// TwinCAT 3 PLC project EDA
// ProgramVersion: 3.1.4024.0
// libraries:
//   Tc2_Standard, * (Beckhoff Automation GmbH)
//   Tc2_System, * (Beckhoff Automation GmbH)
//   Tc3_Module, * (Beckhoff Automation GmbH)
// project tree:
//   GVLs/ GVL.TcGVL
//   / PlcTask.TcTTO
//   POUs/ MAIN.TcPOU
// real-time tasks:
//   TASK PlcTask: cycle T#10ms, priority 20, ADS port 350
// I/O:
//   DEVICE Device 1 (EtherCAT), AmsNetId 5.119.159.52.2.1
//     Term 1 (EK1200) [EK1200-5000 EtherCAT Power supply (2A E-Bus)]
//       Term 2 (EL3443) [EL3443 3Ch. Power Measuring]
//       Term 3 (EL9011) [EL9011 End Terminal]
// variable links:
//   EDA/EDA Instance <-> Device 1 (EtherCAT)/Term 1 (EK1200)/Term 2 (EL3443)
//     PlcTask Inputs/GVL.EL3443.MDP5001_341_Input/MDP5001_341_L1_Basic_Current <-> L1 Basic/Current
//     PlcTask Inputs/GVL.EL3443.MDP5001_341_Input/MDP5001_341_L1_Basic_Voltage <-> L1 Basic/Voltage
//     PlcTask Inputs/GVL.EL3443.MDP5001_341_Input/MDP5001_341_L1_Power_Active_Power <-> L1 Power/Active Power
//     PlcTask Inputs/GVL.EL3443.MDP5001_341_Input/MDP5001_341_L1_Power_Apparent_Power <-> L1 Power/Apparent Power
//     PlcTask Inputs/GVL.EL3443.MDP5001_341_Input/MDP5001_341_L1_Power_Power_Factor <-> L1 Power/Power Factor
//     PlcTask Inputs/GVL.EL3443.MDP5001_341_Input/MDP5001_341_L1_Power_Reactive_Power <-> L1 Power/Reactive Power
//     PlcTask Inputs/GVL.EL3443.MDP5001_341_Input/MDP5001_341_L1_Status_Current_Guard_Error <-> L1 Status/Current Guard Error
//     PlcTask Inputs/GVL.EL3443.MDP5001_341_Input/MDP5001_341_L1_Status_Current_Guard_Warning <-> L1 Status/Current Guard Warning
//     PlcTask Inputs/GVL.EL3443.MDP5001_341_Input/MDP5001_341_L1_Status_Inaccurate_Current <-> L1 Status/Inaccurate Current
//     PlcTask Inputs/GVL.EL3443.MDP5001_341_Input/MDP5001_341_L1_Status_Inaccurate_Voltage <-> L1 Status/Inaccurate Voltage
//     PlcTask Inputs/GVL.EL3443.MDP5001_341_Input/MDP5001_341_L1_Status_Overcurrent <-> L1 Status/Overcurrent
//     PlcTask Inputs/GVL.EL3443.MDP5001_341_Input/MDP5001_341_L1_Status_Overvoltage <-> L1 Status/Overvoltage
//     PlcTask Inputs/GVL.EL3443.MDP5001_341_Input/MDP5001_341_L1_Status_TxPDO_Toggle <-> L1 Status/TxPDO Toggle
//     PlcTask Inputs/GVL.EL3443.MDP5001_341_Input/MDP5001_341_L1_Status_Voltage_Guard_Error <-> L1 Status/Voltage Guard Error
//     PlcTask Inputs/GVL.EL3443.MDP5001_341_Input/MDP5001_341_L1_Status_Voltage_Guard_Warning <-> L1 Status/Voltage Guard Warning
//     PlcTask Inputs/GVL.EL3443.MDP5001_341_Input/MDP5001_341_L1_Status_Voltage_Sign_Bit <-> L1 Status/Voltage Sign Bit
//     PlcTask Inputs/GVL.EL3443.MDP5001_341_Input/MDP5001_341_L1_Timing_Voltage_Last_Zero_Crossing <-> L1 Timing/Voltage Last Zero Crossing
//     PlcTask Inputs/GVL.EL3443.MDP5001_341_Input/MDP5001_341_Total_Basic_Calculated_Neutral_Line_Current <-> Total Basic/Calculated Neutral Line Current
//     PlcTask Inputs/GVL.EL3443.MDP5001_341_Input/MDP5001_341_Total_Basic_Frequency <-> Total Basic/Frequency
//     PlcTask Inputs/GVL.EL3443.MDP5001_341_Input/MDP5001_341_Total_Basic_Power_Factor <-> Total Basic/Power Factor
//     PlcTask Inputs/GVL.EL3443.MDP5001_341_Input/MDP5001_341_Total_Status_Active_Power_Guard_Error <-> Total Status/Active Power Guard Error
//     PlcTask Inputs/GVL.EL3443.MDP5001_341_Input/MDP5001_341_Total_Status_Active_Power_Guard_Warning <-> Total Status/Active Power Guard Warning
//     PlcTask Inputs/GVL.EL3443.MDP5001_341_Input/MDP5001_341_Total_Status_Apparent_Power_Guard_Error <-> Total Status/Apparent Power Guard Error
//     PlcTask Inputs/GVL.EL3443.MDP5001_341_Input/MDP5001_341_Total_Status_Apparent_Power_Guard_Warning <-> Total Status/Apparent Power Guard Warning
//     PlcTask Inputs/GVL.EL3443.MDP5001_341_Input/MDP5001_341_Total_Status_Frequency_Guard_Error <-> Total Status/Frequency Guard Error
//     PlcTask Inputs/GVL.EL3443.MDP5001_341_Input/MDP5001_341_Total_Status_Frequency_Guard_Warning <-> Total Status/Frequency Guard Warning
//     PlcTask Inputs/GVL.EL3443.MDP5001_341_Input/MDP5001_341_Total_Status_Grid_Direction <-> Total Status/Grid Direction
//     PlcTask Inputs/GVL.EL3443.MDP5001_341_Input/MDP5001_341_Total_Status_Neutral_Current_Guard_Error <-> Total Status/Neutral Current Guard Error
//     PlcTask Inputs/GVL.EL3443.MDP5001_341_Input/MDP5001_341_Total_Status_Neutral_Current_Guard_Warning <-> Total Status/Neutral Current Guard Warning
//     PlcTask Inputs/GVL.EL3443.MDP5001_341_Input/MDP5001_341_Total_Status_Power_Quality_Factor <-> Total Status/Power Quality Factor
//     PlcTask Inputs/GVL.EL3443.MDP5001_341_Input/MDP5001_341_Total_Status_Power_Quality_Guard_Error <-> Total Status/Power Quality Guard Error
//     PlcTask Inputs/GVL.EL3443.MDP5001_341_Input/MDP5001_341_Total_Status_Power_Quality_Guard_Warning <-> Total Status/Power Quality Guard Warning
//     PlcTask Inputs/GVL.EL3443.MDP5001_341_Input/MDP5001_341_Total_Status_System_State <-> Total Status/System State
//     PlcTask Inputs/GVL.EL3443.MDP5001_341_Input/MDP5001_341_Total_Status_TxPDO_State <-> Total Status/TxPDO State
//     PlcTask Inputs/GVL.EL3443.MDP5001_341_Input/MDP5001_341_Total_Status_TxPDO_Toggle <-> Total Status/TxPDO Toggle

CONFIGURATION EDA
    RESOURCE PLC ON TwinCAT3
        TASK PlcTask(INTERVAL := T#10ms, PRIORITY := 20);
        PROGRAM MAIN WITH PlcTask : MAIN;
    END_RESOURCE
END_CONFIGURATION

// ---- GVLs/GVL.TcGVL
{attribute 'qualified_only'}
VAR_GLOBAL
	EL3443	:	MDP5001_341_16F33964;
END_VAR

// ---- POUs/MAIN.TcPOU
PROGRAM MAIN
VAR
	
END_VAR

END_PROGRAM
